Fanuc KAREL source: kf00115.KL

-- PROVISIONAL review KL for V1013-1; original PC SHA256 b7b5386f0f6efabba9b53042bd2f2f74b1b74bec25bb50881842370e0167f31b
-- Incomplete behavior may be omitted. Consult companion uncertainty JSON. Do not deploy.
PROGRAM KF00115
%NOLOCKGROUP
BEGIN
  -- UNRESOLVED_PC offsets 0-1; opcodes 7B
  -- UNRESOLVED_PC offsets 6-18; opcodes 2D,9D,52,7F
  -- UNRESOLVED_PC offsets 23-27; opcodes 7F
  -- UNRESOLVED_PC offsets 32-48; opcodes 27,27,2E,AA,23
  -- UNRESOLVED_PC offsets 53-57; opcodes 7F
END KF00115
